% RSLogix 500 project Job 13 part 2 - Leo Kniffen.RSS, saved by version 10.00.00.00 %
PROJECT "ML04B"    % processor: Bul.1763 MicroLogix 1100 Series B %

PROGRAM FILES
  LAD 2   12 rungs

DATA FILES
  O0 OUTPUT  4 elements
  I1 INPUT  6 elements
  S2 STATUS  66 elements
  B3 BINARY  1 elements
  T4 TIMER  1 elements
  C5 COUNTER  1 elements
  R6 CONTROL  1 elements
  N7 INTEGER  1 elements
  F8 FLOAT  1 elements

LADDER 2
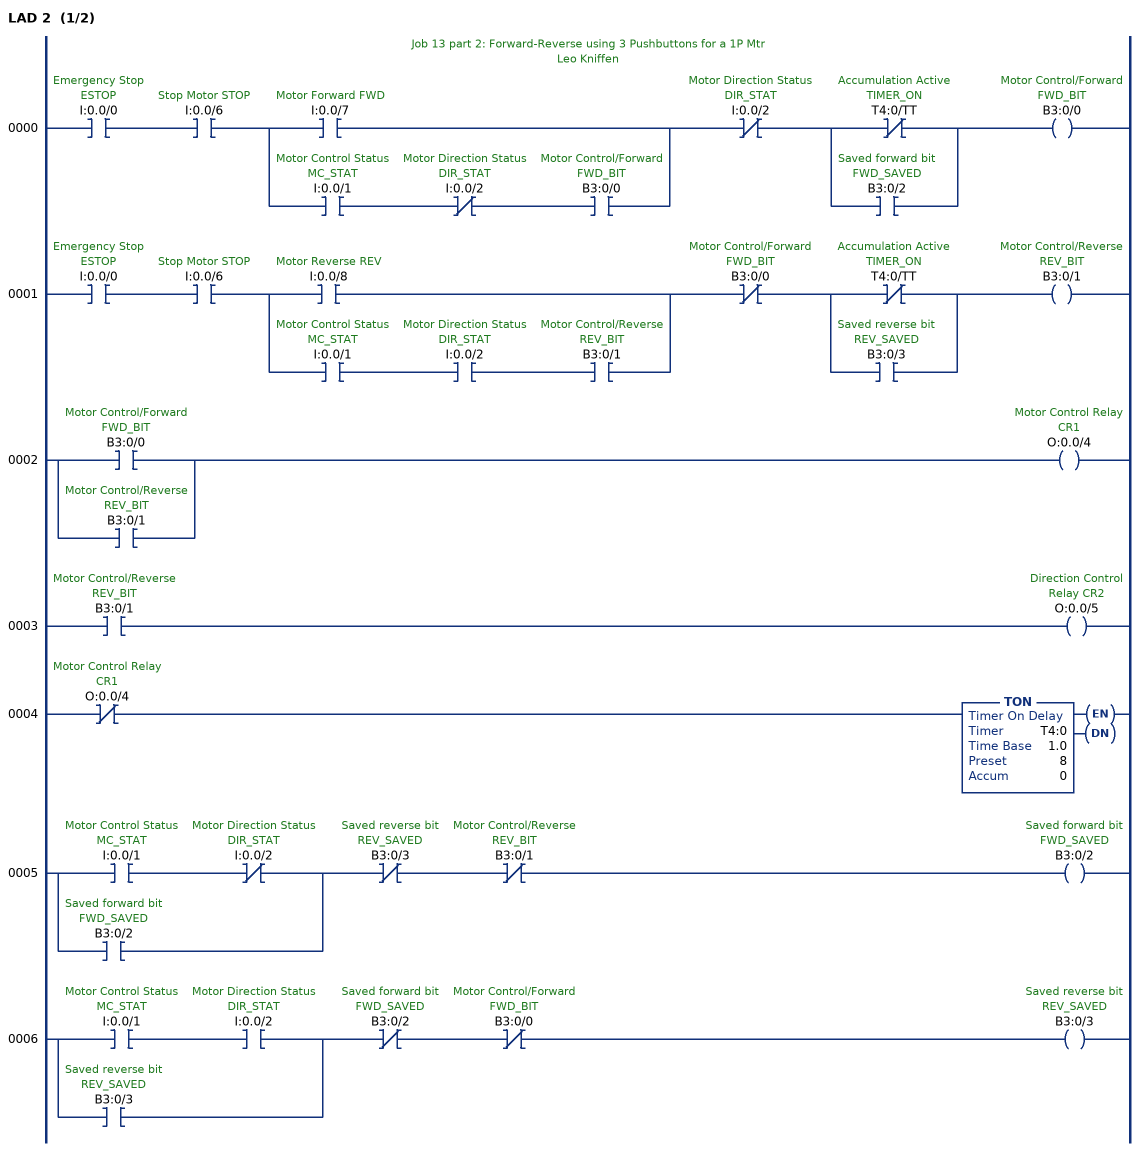
% Rung: 0 %
% Job 13 part 2: Forward-Reverse using 3 Pushbuttons for a 1P Mtr
% Leo Kniffen %
SOR XIC I:0.0/0 XIC I:0.0/6 BST XIC I:0.0/7 NXB XIC I:0.0/1 XIO I:0.0/2 XIC B3:0/0 BND XIO I:0.0/2 BST XIO T4:0/TT NXB XIC B3:0/2 BND OTE B3:0/0 EOR
%   I:0.0/0  ESTOP  "Emergency Stop" %
%   I:0.0/6  STOP  "Stop Motor" %
%   I:0.0/7  FWD  "Motor Forward" %
%   I:0.0/1  MC_STAT  "Motor Control Status" %
%   I:0.0/2  DIR_STAT  "Motor Direction Status" %
%   B3:0/0  FWD_BIT  "Motor Control/Forward" %
%   T4:0/TT  TIMER_ON  "Accumulation Active" %
%   B3:0/2  FWD_SAVED  "Saved forward bit" %
% Rung: 1 %
SOR XIC I:0.0/0 XIC I:0.0/6 BST XIC I:0.0/8 NXB XIC I:0.0/1 XIC I:0.0/2 XIC B3:0/1 BND XIO B3:0/0 BST XIO T4:0/TT NXB XIC B3:0/3 BND OTE B3:0/1 EOR
%   I:0.0/0  ESTOP  "Emergency Stop" %
%   I:0.0/6  STOP  "Stop Motor" %
%   I:0.0/8  REV  "Motor Reverse" %
%   I:0.0/1  MC_STAT  "Motor Control Status" %
%   I:0.0/2  DIR_STAT  "Motor Direction Status" %
%   B3:0/1  REV_BIT  "Motor Control/Reverse" %
%   B3:0/0  FWD_BIT  "Motor Control/Forward" %
%   T4:0/TT  TIMER_ON  "Accumulation Active" %
%   B3:0/3  REV_SAVED  "Saved reverse bit" %
% Rung: 2 %
SOR BST XIC B3:0/0 NXB XIC B3:0/1 BND OTE O:0.0/4 EOR
%   B3:0/0  FWD_BIT  "Motor Control/Forward" %
%   B3:0/1  REV_BIT  "Motor Control/Reverse" %
%   O:0.0/4  CR1  "Motor Control Relay" %
% Rung: 3 %
SOR XIC B3:0/1 OTE O:0.0/5 EOR
%   B3:0/1  REV_BIT  "Motor Control/Reverse" %
%   O:0.0/5  CR2  "Direction Control Relay" %
% Rung: 4 %
SOR XIO O:0.0/4 TON T4:0 1.0 8 0 EOR
%   O:0.0/4  CR1  "Motor Control Relay" %
% Rung: 5 %
SOR BST XIC I:0.0/1 XIO I:0.0/2 NXB XIC B3:0/2 BND XIO B3:0/3 XIO B3:0/1 OTE B3:0/2 EOR
%   I:0.0/1  MC_STAT  "Motor Control Status" %
%   I:0.0/2  DIR_STAT  "Motor Direction Status" %
%   B3:0/2  FWD_SAVED  "Saved forward bit" %
%   B3:0/3  REV_SAVED  "Saved reverse bit" %
%   B3:0/1  REV_BIT  "Motor Control/Reverse" %
% Rung: 6 %
SOR BST XIC I:0.0/1 XIC I:0.0/2 NXB XIC B3:0/3 BND XIO B3:0/2 XIO B3:0/0 OTE B3:0/3 EOR
%   I:0.0/1  MC_STAT  "Motor Control Status" %
%   I:0.0/2  DIR_STAT  "Motor Direction Status" %
%   B3:0/3  REV_SAVED  "Saved reverse bit" %
%   B3:0/2  FWD_SAVED  "Saved forward bit" %
%   B3:0/0  FWD_BIT  "Motor Control/Forward" %

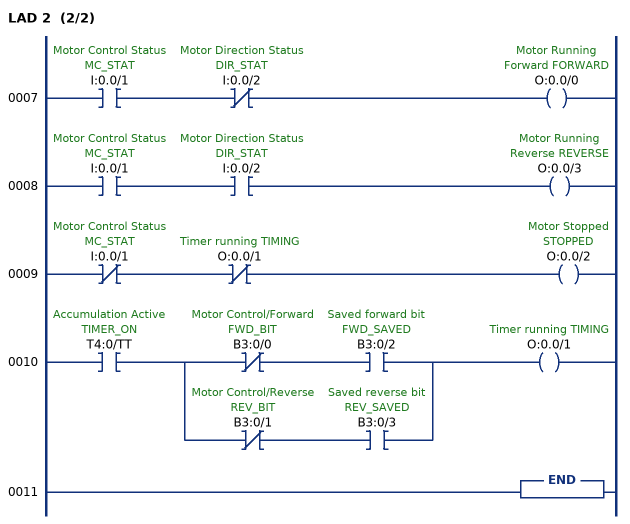
% Rung: 7 %
SOR XIC I:0.0/1 XIO I:0.0/2 OTE O:0.0/0 EOR
%   I:0.0/1  MC_STAT  "Motor Control Status" %
%   I:0.0/2  DIR_STAT  "Motor Direction Status" %
%   O:0.0/0  FORWARD  "Motor Running Forward" %
% Rung: 8 %
SOR XIC I:0.0/1 XIC I:0.0/2 OTE O:0.0/3 EOR
%   I:0.0/1  MC_STAT  "Motor Control Status" %
%   I:0.0/2  DIR_STAT  "Motor Direction Status" %
%   O:0.0/3  REVERSE  "Motor Running Reverse" %
% Rung: 9 %
SOR XIO I:0.0/1 XIO O:0.0/1 OTE O:0.0/2 EOR
%   I:0.0/1  MC_STAT  "Motor Control Status" %
%   O:0.0/1  TIMING  "Timer running" %
%   O:0.0/2  STOPPED  "Motor Stopped" %
% Rung: 10 %
SOR XIC T4:0/TT BST XIO B3:0/0 XIC B3:0/2 NXB XIO B3:0/1 XIC B3:0/3 BND OTE O:0.0/1 EOR
%   T4:0/TT  TIMER_ON  "Accumulation Active" %
%   B3:0/0  FWD_BIT  "Motor Control/Forward" %
%   B3:0/2  FWD_SAVED  "Saved forward bit" %
%   B3:0/1  REV_BIT  "Motor Control/Reverse" %
%   B3:0/3  REV_SAVED  "Saved reverse bit" %
%   O:0.0/1  TIMING  "Timer running" %
% Rung: 11 %
SOR END EOR

OTHER DOCUMENTED ADDRESSES
  I:0.0/3  DIRECTION_FWD  "Direction: Forward- Off-Reverse"
  I:0.0/4  DIRECTION_REV  "Direction: Forward- Off-Reverse"
  I:0.0/5  RUN_JOG  "Run/Jog Mode (A=Run, B=Jog)"
  T4:0/DN  TIMER_D  "Timer Done"
  T4:0/EN  TIMER_E  "Timer enable"

DATA TABLE (non-zero values as saved)
DATA T4
% .PRE .ACC %
% T4:0 % 8 0
